PROGRAM TestMain
VAR
  test_assert: TestAssert;
  test_sbo: TestStringBufferOutput;
END_VAR

test_assert();
test_sbo();

END_PROGRAM

(* stored: Version 1.1.0.1, ProductVersion 3.1.4022.7
   POU TestMain: Id {d4bce498-62ef-4564-9c96-addc02b4bbba}, SpecialFunc None *)
